// Mitsubishi GX Developer project: plcABCplc课程设计梯形图-四层电梯   PLC: FX2N

PROGRAM MAIN
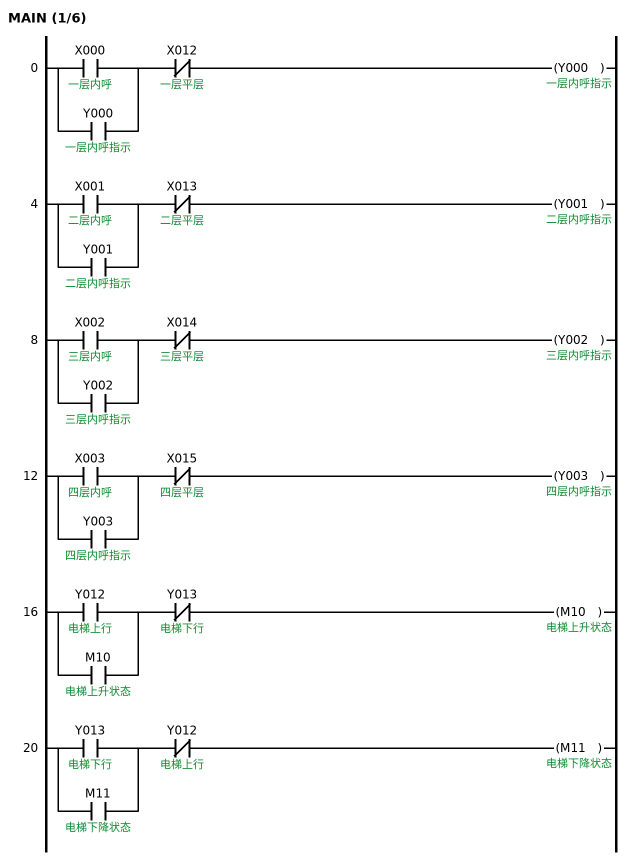
0     LD      X000  ; 一层内呼
      OR      Y000  ; 一层内呼指示
      ANI     X012  ; 一层平层
      OUT     Y000  ; 一层内呼指示
4     LD      X001  ; 二层内呼
      OR      Y001  ; 二层内呼指示
      ANI     X013  ; 二层平层
      OUT     Y001  ; 二层内呼指示
8     LD      X002  ; 三层内呼
      OR      Y002  ; 三层内呼指示
      ANI     X014  ; 三层平层
      OUT     Y002  ; 三层内呼指示
12    LD      X003  ; 四层内呼
      OR      Y003  ; 四层内呼指示
      ANI     X015  ; 四层平层
      OUT     Y003  ; 四层内呼指示
16    LD      Y012  ; 电梯上行
      OR      M10  ; 电梯上升状态
      ANI     Y013  ; 电梯下行
      OUT     M10  ; 电梯上升状态
20    LD      Y013  ; 电梯下行
      OR      M11  ; 电梯下降状态
      ANI     Y012  ; 电梯上行
      OUT     M11  ; 电梯下降状态
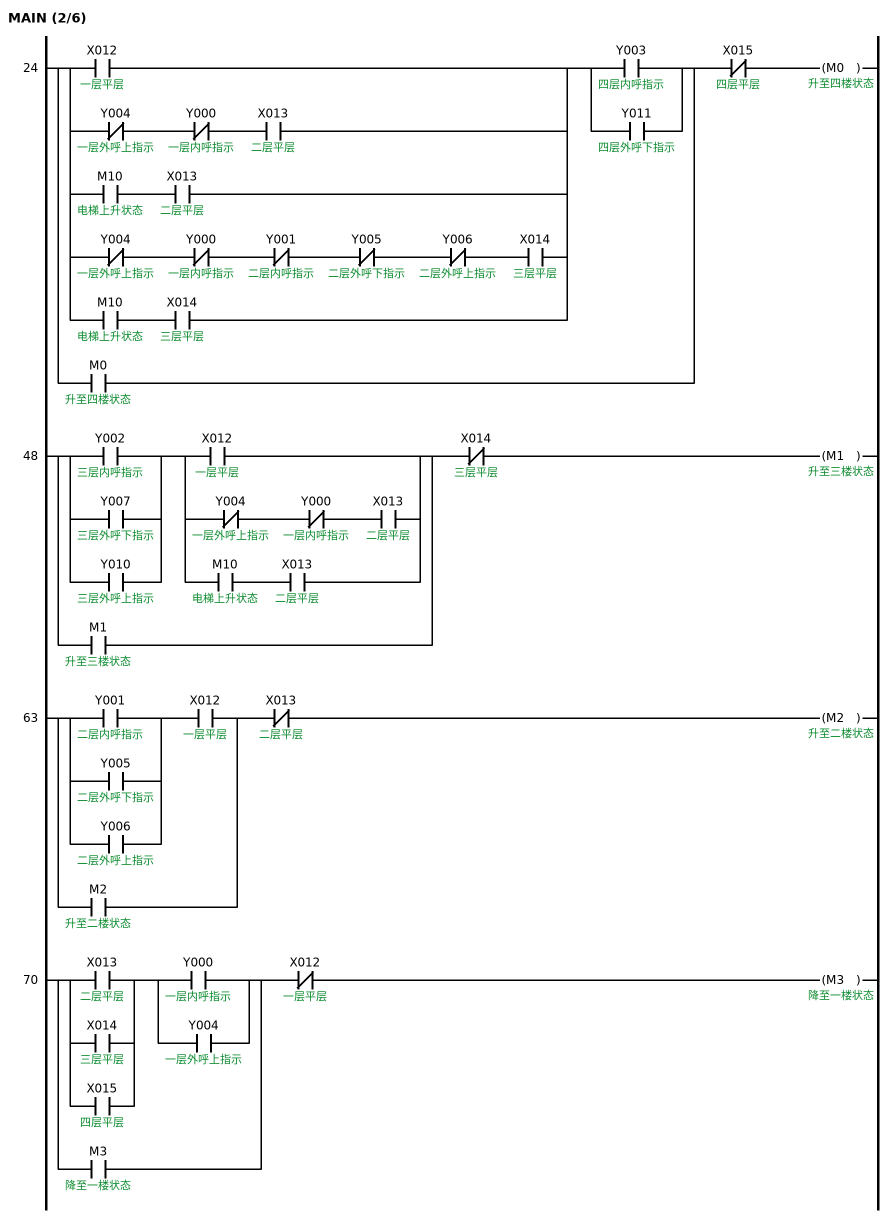
24    LD      X012  ; 一层平层
      LDI     Y004  ; 一层外呼上指示
      ANI     Y000  ; 一层内呼指示
      AND     X013  ; 二层平层
      ORB
      LD      M10  ; 电梯上升状态
      AND     X013  ; 二层平层
      ORB
      LDI     Y004  ; 一层外呼上指示
      ANI     Y000  ; 一层内呼指示
      ANI     Y001  ; 二层内呼指示
      ANI     Y005  ; 二层外呼下指示
      ANI     Y006  ; 二层外呼上指示
      AND     X014  ; 三层平层
      ORB
      LD      M10  ; 电梯上升状态
      AND     X014  ; 三层平层
      ORB
      LD      Y003  ; 四层内呼指示
      OR      Y011  ; 四层外呼下指示
      ANB
      OR      M0  ; 升至四楼状态
      ANI     X015  ; 四层平层
      OUT     M0  ; 升至四楼状态
48    LD      Y002  ; 三层内呼指示
      OR      Y007  ; 三层外呼下指示
      OR      Y010  ; 三层外呼上指示
      LD      X012  ; 一层平层
      LDI     Y004  ; 一层外呼上指示
      ANI     Y000  ; 一层内呼指示
      AND     X013  ; 二层平层
      ORB
      LD      M10  ; 电梯上升状态
      AND     X013  ; 二层平层
      ORB
      ANB
      OR      M1  ; 升至三楼状态
      ANI     X014  ; 三层平层
      OUT     M1  ; 升至三楼状态
63    LD      Y001  ; 二层内呼指示
      OR      Y005  ; 二层外呼下指示
      OR      Y006  ; 二层外呼上指示
      AND     X012  ; 一层平层
      OR      M2  ; 升至二楼状态
      ANI     X013  ; 二层平层
      OUT     M2  ; 升至二楼状态
70    LD      X013  ; 二层平层
      OR      X014  ; 三层平层
      OR      X015  ; 四层平层
      LD      Y000  ; 一层内呼指示
      OR      Y004  ; 一层外呼上指示
      ANB
      OR      M3  ; 降至一楼状态
      ANI     X012  ; 一层平层
      OUT     M3  ; 降至一楼状态
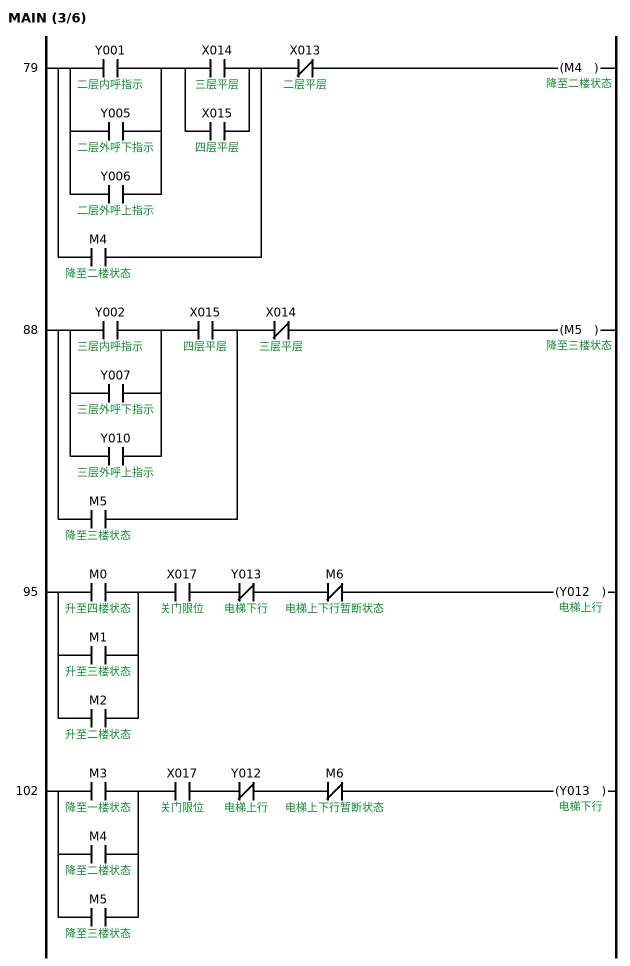
79    LD      Y001  ; 二层内呼指示
      OR      Y005  ; 二层外呼下指示
      OR      Y006  ; 二层外呼上指示
      LD      X014  ; 三层平层
      OR      X015  ; 四层平层
      ANB
      OR      M4  ; 降至二楼状态
      ANI     X013  ; 二层平层
      OUT     M4  ; 降至二楼状态
88    LD      Y002  ; 三层内呼指示
      OR      Y007  ; 三层外呼下指示
      OR      Y010  ; 三层外呼上指示
      AND     X015  ; 四层平层
      OR      M5  ; 降至三楼状态
      ANI     X014  ; 三层平层
      OUT     M5  ; 降至三楼状态
95    LD      M0  ; 升至四楼状态
      OR      M1  ; 升至三楼状态
      OR      M2  ; 升至二楼状态
      AND     X017  ; 关门限位
      ANI     Y013  ; 电梯下行
      ANI     M6  ; 电梯上下行暂断状态
      OUT     Y012  ; 电梯上行
102   LD      M3  ; 降至一楼状态
      OR      M4  ; 降至二楼状态
      OR      M5  ; 降至三楼状态
      AND     X017  ; 关门限位
      ANI     Y012  ; 电梯上行
      ANI     M6  ; 电梯上下行暂断状态
      OUT     Y013  ; 电梯下行
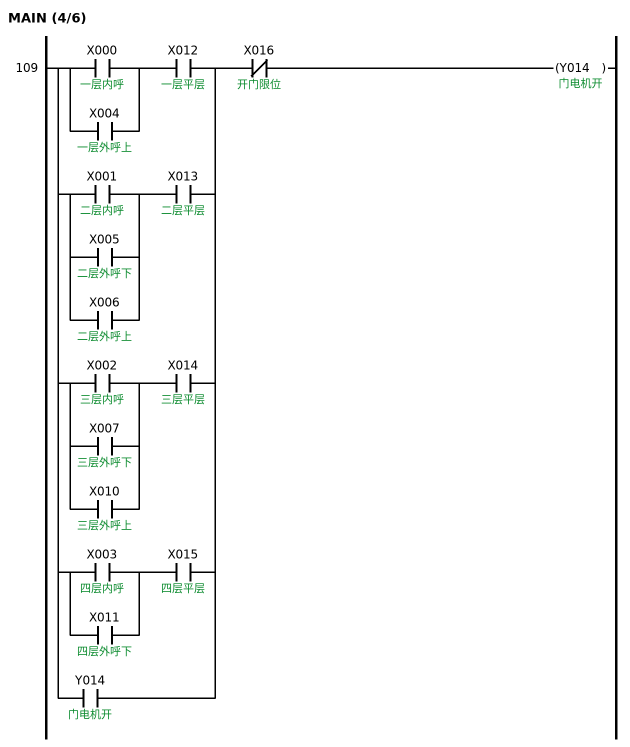
109   LD      X000  ; 一层内呼
      OR      X004  ; 一层外呼上
      AND     X012  ; 一层平层
      LD      X001  ; 二层内呼
      OR      X005  ; 二层外呼下
      OR      X006  ; 二层外呼上
      AND     X013  ; 二层平层
      ORB
      LD      X002  ; 三层内呼
      OR      X007  ; 三层外呼下
      OR      X010  ; 三层外呼上
      AND     X014  ; 三层平层
      ORB
      LD      X003  ; 四层内呼
      OR      X011  ; 四层外呼下
      AND     X015  ; 四层平层
      ORB
      OR      Y014  ; 门电机开
      ANI     X016  ; 开门限位
      OUT     Y014  ; 门电机开
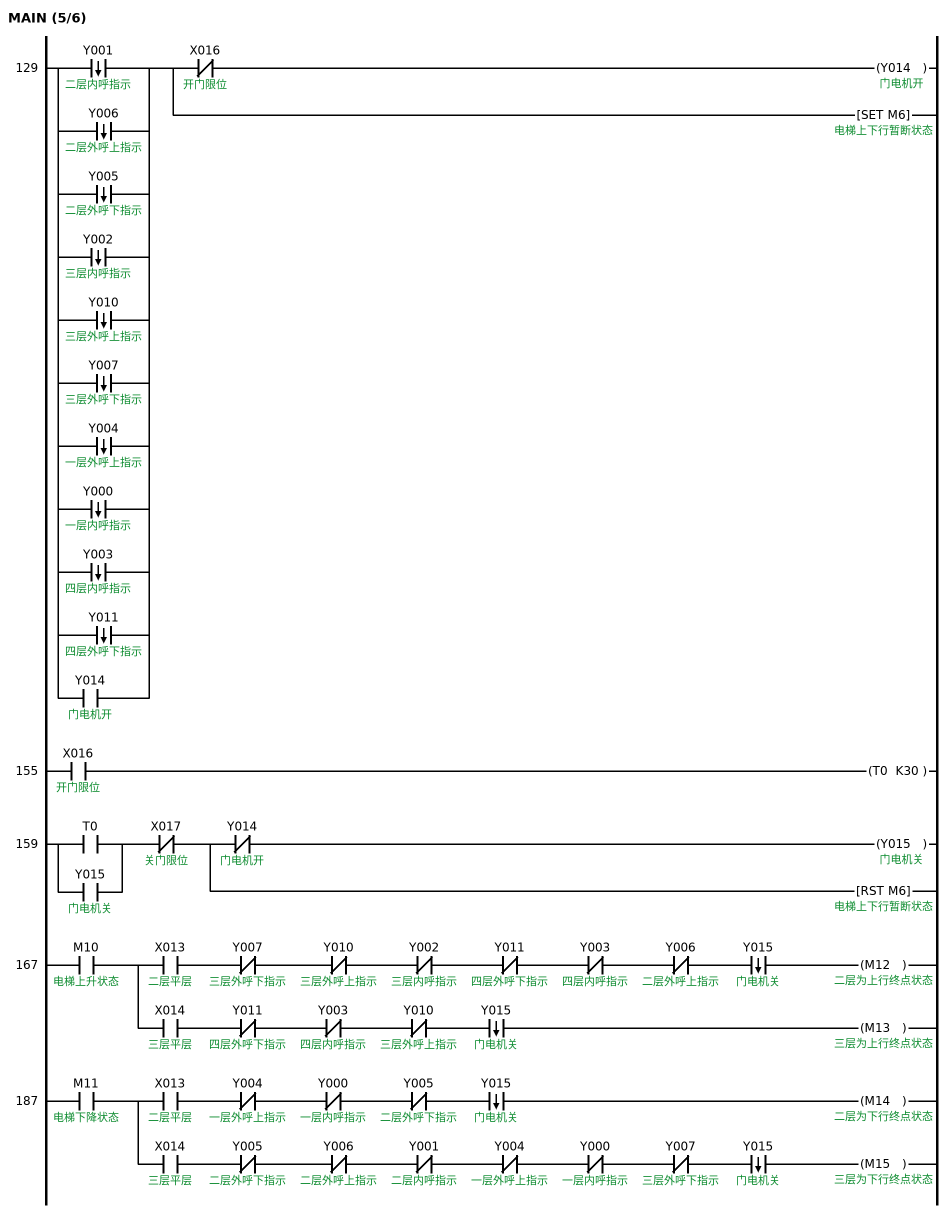
129   LDF     Y001  ; 二层内呼指示
      ORF     Y006  ; 二层外呼上指示
      ORF     Y005  ; 二层外呼下指示
      ORF     Y002  ; 三层内呼指示
      ORF     Y010  ; 三层外呼上指示
      ORF     Y007  ; 三层外呼下指示
      ORF     Y004  ; 一层外呼上指示
      ORF     Y000  ; 一层内呼指示
      ORF     Y003  ; 四层内呼指示
      ORF     Y011  ; 四层外呼下指示
      OR      Y014  ; 门电机开
      MPS
      ANI     X016  ; 开门限位
      OUT     Y014  ; 门电机开
      MPP
      SET     M6  ; 电梯上下行暂断状态
155   LD      X016  ; 开门限位
      OUT     T0 K30
159   LD      T0
      OR      Y015  ; 门电机关
      ANI     X017  ; 关门限位
      MPS
      ANI     Y014  ; 门电机开
      OUT     Y015  ; 门电机关
      MPP
      RST     M6  ; 电梯上下行暂断状态
167   LD      M10  ; 电梯上升状态
      MPS
      AND     X013  ; 二层平层
      ANI     Y007  ; 三层外呼下指示
      ANI     Y010  ; 三层外呼上指示
      ANI     Y002  ; 三层内呼指示
      ANI     Y011  ; 四层外呼下指示
      ANI     Y003  ; 四层内呼指示
      ANI     Y006  ; 二层外呼上指示
      ANDF    Y015  ; 门电机关
      OUT     M12  ; 二层为上行终点状态
      MPP
      AND     X014  ; 三层平层
      ANI     Y011  ; 四层外呼下指示
      ANI     Y003  ; 四层内呼指示
      ANI     Y010  ; 三层外呼上指示
      ANDF    Y015  ; 门电机关
      OUT     M13  ; 三层为上行终点状态
187   LD      M11  ; 电梯下降状态
      MPS
      AND     X013  ; 二层平层
      ANI     Y004  ; 一层外呼上指示
      ANI     Y000  ; 一层内呼指示
      ANI     Y005  ; 二层外呼下指示
      ANDF    Y015  ; 门电机关
      OUT     M14  ; 二层为下行终点状态
      MPP
      AND     X014  ; 三层平层
      ANI     Y005  ; 二层外呼下指示
      ANI     Y006  ; 二层外呼上指示
      ANI     Y001  ; 二层内呼指示
      ANI     Y004  ; 一层外呼上指示
      ANI     Y000  ; 一层内呼指示
      ANI     Y007  ; 三层外呼下指示
      ANDF    Y015  ; 门电机关
      OUT     M15  ; 三层为下行终点状态
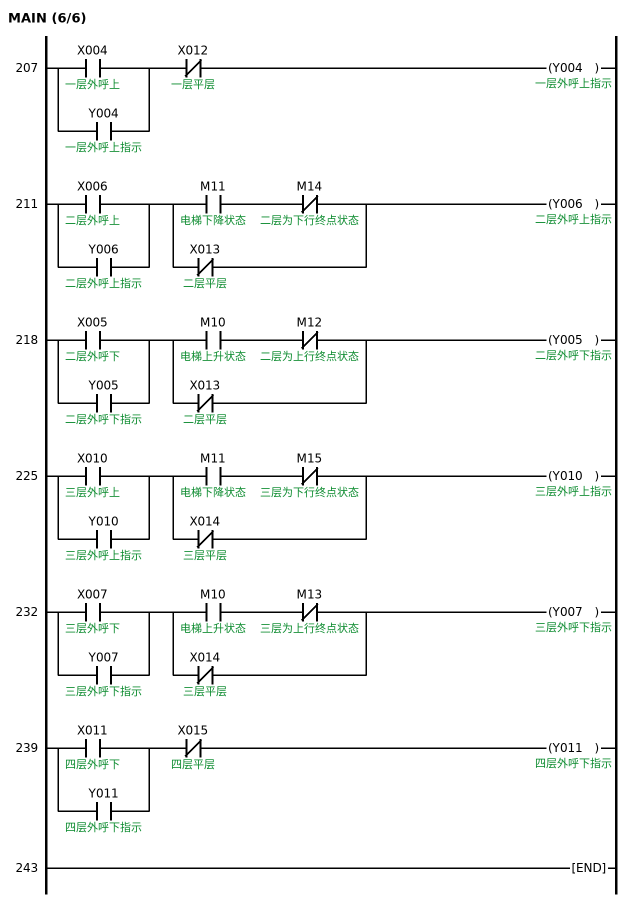
207   LD      X004  ; 一层外呼上
      OR      Y004  ; 一层外呼上指示
      ANI     X012  ; 一层平层
      OUT     Y004  ; 一层外呼上指示
211   LD      X006  ; 二层外呼上
      OR      Y006  ; 二层外呼上指示
      LD      M11  ; 电梯下降状态
      ANI     M14  ; 二层为下行终点状态
      ORI     X013  ; 二层平层
      ANB
      OUT     Y006  ; 二层外呼上指示
218   LD      X005  ; 二层外呼下
      OR      Y005  ; 二层外呼下指示
      LD      M10  ; 电梯上升状态
      ANI     M12  ; 二层为上行终点状态
      ORI     X013  ; 二层平层
      ANB
      OUT     Y005  ; 二层外呼下指示
225   LD      X010  ; 三层外呼上
      OR      Y010  ; 三层外呼上指示
      LD      M11  ; 电梯下降状态
      ANI     M15  ; 三层为下行终点状态
      ORI     X014  ; 三层平层
      ANB
      OUT     Y010  ; 三层外呼上指示
232   LD      X007  ; 三层外呼下
      OR      Y007  ; 三层外呼下指示
      LD      M10  ; 电梯上升状态
      ANI     M13  ; 三层为上行终点状态
      ORI     X014  ; 三层平层
      ANB
      OUT     Y007  ; 三层外呼下指示
239   LD      X011  ; 四层外呼下
      OR      Y011  ; 四层外呼下指示
      ANI     X015  ; 四层平层
      OUT     Y011  ; 四层外呼下指示
243   END
END_PROGRAM
